# B&R Automation Studio project RS15_RX_30005_r00 (part 6)

#### BackUpCyclic.st - Cyclic code
```iecst
(********************************************************************
 * COPYRIGHT --
 ********************************************************************
 * Program: BackUp
 * File: BackUpCyclic.st
 * Author: pkiel
 * Created: December 11, 2009
 ********************************************************************
 * Implementation of program BackUp
 ********************************************************************)

PROGRAM _CYCLIC

	TON_0(IN := SystemBackUp_PB, PT := T#5s); 	(* Trigger File Write *)
	TON_1(IN := SystemRestore_PB, PT := T#5s); 	(* Trigger File Read *)
	TON_2(IN := NOT(bOK), PT := T#5s); 			(* Error Timer *)
	TON_3(IN := OpComplete, PT := T#5s); 		(* Operation Complete Timer *)
	TON_4(IN := FileNotFound, PT := T#5s); 		(* File Not Found Timer *)

	CASE byStep OF

			0: (**** Loop For Command Selection ****)

					IF (EDGEPOS(TON_0.Q)) THEN
						cmdSystemBackUp := 1;
						byStep := 1;
					ELSIF (EDGEPOS(TON_1.Q)) THEN
	                	cmdSystemRestore := 1;
						byStep := 1;
					END_IF

			1: (**** Try to open existing file ****)
	                (* Initialize file open structrue *)
	                FOpen.enable    := 1;
	                FOpen.pDevice   := ADR(strDevice);
	                FOpen.pFile     := ADR(strFile);
	                FOpen.mode      := FILE_RW;  (* Read and write access *)

	                (* Call FBK *)
	                FOpen();

	                (* Get FBK output information *)
	                dwIdent := FOpen.ident;
	                wStatus := FOpen.status;

	                (* Verify status (20708 -> File doesn't exist) *)
	                IF (wStatus = 20708) THEN
	                        IF cmdSystemBackUp THEN
									byStep := 2;
							ELSIF cmdSystemRestore THEN
	                        		byStep := 11;
							END_IF
	                ELSE
	                        IF (wStatus = 0) THEN
	                            IF cmdSystemBackUp THEN
									byStep := 3;
								ELSIF cmdSystemRestore THEN
	                        		byStep := 4;
								END_IF
	                        ELSE
	                                IF (wStatus <> 65535) THEN
	                                        byErrorLevel := 1;
	                                        byStep := 10;

	                                        IF (wStatus = 20799) THEN
	                                                wError := FileIoGetSysError();
	                                        END_IF
	                                END_IF
	                        END_IF
	                END_IF

	        2: (**** Create file ****)
	                (* Initialize file create structure *)
	                FCreate.enable  := 1;
	                FCreate.pDevice := ADR(strDevice);
	                FCreate.pFile   := ADR(strFile);

	                (* Call FBK *)
	                FCreate();

	                (* Get FBK output information *)
	                dwIdent := FCreate.ident;
	                wStatus := FCreate.status;

	                (* Verify status *)
	                IF (wStatus = 0) THEN
							byStep := 3;
	                ELSE
	                        IF (wStatus <> 65535) THEN
	                                byErrorLevel := 2;
	                                byStep := 10;

	                                IF (wStatus = 20799) THEN
	                                        wError := FileIoGetSysError();
	                                END_IF
	                        END_IF
	                END_IF

	        3: (**** Write data to file ****)
	                (* Load Data Into System Structure *)
					SystemData.gSP_A	 				        := gSP_A;
					SystemData.gReg 					        := gReg;
					SystemData.gPassword 				      := gPassword;
					SystemData.gMachineTime				    := gMachineTime;
					SystemData.gSP_CmdSpeed				    := gSP_CmdSpeed;
					SystemData.gSP_ColdGlue				    := gSP_ColdGlue;
					SystemData.gSP_HotGlue				    := gSP_HotGlue;
					SystemData.gSP_GlueTrayAutoSpeed	:= gSP_GlueTrayAutoSpeed;
					SystemData.gSP_PerfCylSelect		  := gSP_PerfCylSelect;
					SystemData.gSP_PerfKnifeCount		  := gSP_PerfKnifeCount;
					SystemData.gSP_TubeSelect		  	  := gSP_TubeSelect;

					(* Write System Structure To File *)
	                FWrite.enable   := 1;
	                FWrite.ident    := dwIdent;
	                FWrite.offset   := 0;
	                FWrite.pSrc     := ADR(SystemData);
	                FWrite.len      := SIZEOF(SystemData);

	                (* Call FBK *)
	                FWrite();

	                (* Get status *)
	                wStatus := FWrite.status;

	                (* Verify status *)
	                IF (wStatus = 0) THEN
	                        byStep := 5;
	                ELSE
	                        IF (wStatus <> 65535) THEN
	                                byErrorLevel := 3;
	                                byStep := 10;

	                                IF (wStatus = 20799) THEN
	                                        wError := FileIoGetSysError();
	                                END_IF
	                        END_IF
	                END_IF

	        4: (**** Read data from file ****)
	                (* Initialize file read structure *)
	                FRead.enable    := 1;
	                FRead.ident     := dwIdent;
	                FRead.offset    := 0;
	                FRead.pDest     := ADR(SystemData);
	                FRead.len       := SIZEOF(SystemData);

	                (* Call FBK *)
	                FRead();

	                (* Get status *)
	                wStatus := FRead.status;

	                (* Verify status *)
	                IF (wStatus = 0) THEN
						gSP_A 						    := SystemData.gSP_A;
						gReg 					      	:= SystemData.gReg;
						gPassword 					  := SystemData.gPassword;
						gMachineTime				  := SystemData.gMachineTime;
						gSP_CmdSpeed				  := SystemData.gSP_CmdSpeed;
						gSP_ColdGlue	 			  := SystemData.gSP_ColdGlue;
						gSP_HotGlue					  := SystemData.gSP_HotGlue;
						gSP_GlueTrayAutoSpeed	:= SystemData.gSP_GlueTrayAutoSpeed;
						gSP_PerfCylSelect			:= SystemData.gSP_PerfCylSelect;
						gSP_PerfKnifeCount		:= SystemData.gSP_PerfKnifeCount;
						gSP_TubeSelect				:= SystemData.gSP_TubeSelect;

						byStep := 5;
	                ELSE
	                    IF (wStatus <> 65535) THEN
	                 	   byErrorLevel := 4;
	                       byStep := 10;

	                       IF (wStatus = 20799) THEN
	                    	   wError := FileIoGetSysError();
	                       END_IF
	                	END_IF
	                END_IF

	        5: (**** Close file ****)
	                (* Initialize file close structure *)
	                FClose.enable   := 1;
	                FClose.ident    := dwIdent;

	                (* Call FBK *)
	                FClose();

	                (* Get status *)
	                wStatus := FClose.status;

	                (* Verify status *)
	                IF (wStatus = 0) THEN
							cmdSystemBackUp := 0;
							cmdSystemRestore := 0;
	                        OpComplete := 1;
							byStep := 6;
	                ELSE
	                        IF (wStatus <> 65535) THEN
	                                byErrorLevel := 5;
	                                byStep := 10;

	                                IF (wStatus = 20799) THEN
	                                        wError := FileIoGetSysError();
	                                END_IF
	                        END_IF
	                END_IF

	        6: (**** Operation Complete ****)

	                IF (TON_3.Q) THEN
						OpComplete := 0;
						byStep := 0;
					END_IF

			10: (**** Error step ****)
	                bOK := FALSE;
					cmdSystemBackUp := 0;
					cmdSystemRestore := 0;
					IF (TON_2.Q) THEN
						bOK := 1;
						byStep := 0;
					END_IF

			11: (**** File Not Found ****)
	                bOK := FALSE;
					FileNotFound := 1;
					cmdSystemBackUp := 0;
					cmdSystemRestore := 0;
	                IF (TON_4.Q) THEN
						FileNotFound := 0;
						bOK := TRUE;
						byStep := 0;
					END_IF

	END_CASE

END_PROGRAM
```

#### BackUp.var - Local variables
```iecst
(********************************************************************
 * COPYRIGHT --
 ********************************************************************
 * Program: BackUp
 * File: BackUp.var
 * Author: pkiel
 * Created: December 11, 2009
 ********************************************************************
 * Local variables of program BackUp
 ********************************************************************)
VAR
	strDevice : STRING[32];
	strFile : STRING[32];
	byStep : USINT;
	FOpen : FileOpen;
	bOK : BOOL;
	dwIdent : UDINT;
	wStatus : UINT;
	byErrorLevel : USINT;
	wError : UINT;
	FCreate : FileCreate;
	FWrite : FileWrite;
	FRead : FileRead;
	FClose : FileClose;
	TON_0 : TON;
	TON_1 : TON;
	TON_2 : TON;
	TON_3 : TON;
	TON_4 : TON;
	OpComplete : BOOL;
	SystemBackUp_PB : BOOL;
	SystemRestore_PB : BOOL;
	cmdSystemBackUp : BOOL;
	cmdSystemRestore : BOOL;
	FileNotFound : BOOL;
	SystemData : System;
END_VAR
```

- Program Logical/HMI/Cmd_Trace (IEC) (no source held here)

### Program Logical/HMI/CPURestart

#### CPURestartCyclic.st
```iecst
(********************************************************************
 * COPYRIGHT -- .
 ********************************************************************
 * Program: CPURestart
 * File: CPURestartCyclic.st
 * Author: dominique
 * Created: March 18, 2012
 ********************************************************************
 * Implementation of program CPURestart
 ********************************************************************)

PROGRAM _CYCLIC

  // Sytem Restart from HMI

  // Cold
  IF HMI_CmdColdRestart THEN
    HMI_CmdColdRestart := 0 ;
    uiRetColdRestart := SYSreset(1, 2) ;
    IF (uiRetColdRestart <> 0) THEN
      HMI_iCRestartStat := uiRetColdRestart ;
    END_IF
  END_IF

  // Warm
  IF HMI_CmdWarmRestart THEN
    HMI_CmdWarmRestart := 0 ;
    uiRetWarmRestart := SYSreset(1, 1) ;
    IF (uiRetWarmRestart <> 0) THEN
      HMI_iWRestartStat := uiRetWarmRestart ;
    END_IF
  END_IF

  // Reset stat
  IF EDGEPOS(gAlarmReset) THEN
    HMI_iCRestartStat := 0 ;
    HMI_iWRestartStat := 0 ;
  END_IF

END_PROGRAM
```

#### CPURestartInit.st
```iecst
(********************************************************************
 * COPYRIGHT -- .
 ********************************************************************
 * Program: CPURestart
 * File: CPURestartInit.st
 * Author: dominique
 * Created: March 18, 2012
 ********************************************************************
 * Implementation of program CPURestart
 ********************************************************************)

PROGRAM _INIT

END_PROGRAM
```

- FreeLock.clm (not shown)

- GreenRed.clm (not shown)

- Sensor.clm (not shown)

- SetCol_1.clm (not shown)

- Arial10pxBold.fninfo (not shown)

- Arial12px.fninfo (not shown)

- Arial9pxBold.fninfo (not shown)

- Arial_12_Bold.fninfo (not shown)

- Arial_12_Bold_Italic.fninfo (not shown)

- Arial_14_Bold_Italic.fninfo (not shown)

- Arial_15_Bold.fninfo (not shown)

- Arial_18_Bold.fninfo (not shown)

- Arial_18_Italic.fninfo (not shown)

- Arial_20_Bold.fninfo (not shown)

- Arial_26_Bold.fninfo (not shown)

- Arial_36_Bold.fninfo (not shown)

- Arial_8_Bold.fninfo (not shown)

- Arial_9_Bold.fninfo (not shown)

- EnvBagPerfSetUp.layer (not shown)

- PasswordChangeAccepted.layer (not shown)

- PasswordConfirm.layer (not shown)

- PerfSpeedCurve_RS15_Perfo1_2_IF.layer (not shown)

- PerfSpeedCurve_RS26_ApPo_520_IF.layer (not shown)

- PerfSpeedCurve_RS26_Perfo1_IF.layer (not shown)

- PopUp_AxisSynchroInProgress.layer (not shown)

- PopUp_ProductCountReset.layer (not shown)

- SetUpHoldTearApPoDrumRS26.layer (not shown)

- StandPerfSetUp.layer (not shown)

- Underlay_Alarms.layer (not shown)

- Underlay_Main.layer (not shown)

- Underlay_Maintenance.layer (not shown)

- Underlay_Setup.layer (not shown)

- ZZZ.layer (not shown)

- TrendData_1.trd (not shown)

- TrendData_2.trd (not shown)

### Program Logical/HMI/HMI_Control

#### HMI_Control.var
```iecst
(********************************************************************
 * COPYRIGHT --
 ********************************************************************
 * Program: HMI_Control
 * File: HMI_Control.var
 * Author: pkiel
 * Created: September 17, 2009
 ********************************************************************
 * Local variables of program HMI_Control
 ********************************************************************)
VAR
	CfgSetDefaultGateway_0 : CfgSetDefaultGateway;
	DataLock_Motion : UINT;
	HMI_ActualVelocity : REAL;
	HMI_AlarmFilterControl : INT;
	HMI_AlarmFilterGroup : INT;
	HMI_AlarmInputStatus : INT;
	HMI_Error : BOOL;
	HMI_ErrorAck : BOOL;
	HMI_ErrorCount : UINT;
	HMI_ErrorID : UINT;
	HMI_ErrorStop : BOOL;
	HMI_ErrorText : ARRAY[0..3] OF STRING[79];
	HMI_Ind_ContinuousMotion : BOOL;
	HMI_Ind_ControllerStatus : BOOL;
	HMI_Ind_DiscreteMotion : BOOL;
	HMI_Ind_Enabled : BOOL;
	HMI_Ind_Homed : BOOL;
	HMI_Ind_InMotion : BOOL;
	HMI_Ind_NetworkInit : BOOL;
	HMI_Ind_SynchronizedMotion : BOOL;
	HMI_Input_DriveEnable : BOOL;
	HMI_Input_Home : BOOL;
	HMI_Input_Trigger1 : BOOL;
	HMI_Input_Trigger2 : BOOL;
	HMI_MainScreenGroup : UINT;
	HMI_MaintenanceScreenGroup : UINT;
	HMI_PositionDeg : REAL;
	HMI_PositionInch : REAL;
	HMI_Screen2Group_Ind : UINT;
	HMI_ScreenGroup_Ind : UINT;
	HMI_SetupScreenGroup : UINT;
	HMI_Status_Ind : UINT;
	HMI_StatusScreenGroup : UINT;
	HMI_bMaxSpeedPerf_PB : BOOL;
	HMI_iSelCurvMaxSpeedPerf : INT;
	HMI_uiCurvVisibl : UINT;
	HMI_uiNeverVisibl : UINT := 1;
	HMI_strMP_UNW_HydroPump : STRING[10];
	HMI_strMP_FP_MotorFan : STRING[10];
	HMI_strMP_FP_SlowRot1 : STRING[10];
	HMI_strMP_FP_SlowRot2 : STRING[10];
	HMI_strMP_FP_SlowRot3 : STRING[10];
	HMI_strMP_FP_SlowRot4 : STRING[10];
	HMI_strMP_FP_SlowRot5 : STRING[10];
	HMI_strMP_FP_SlowRot6 : STRING[10];
	HMI_strMP_GlueSlowRotation : STRING[10];
	HMI_strMP_PerfFan : STRING[10];
	HMI_strMP_Vacuum : STRING[10];
	HMI_strMP_3W_MotorFan : STRING[10];
	HMI_strMP_DRY_Blower : STRING[12];
	HMI_strMP_DRY_Heater : STRING[10];
	HMI_strSS_DRY_Thermostat : STRING[10];
	HMI_strMP_CMP_WasteSuc : STRING[10];
	HMI_strMP_EB_WasteSuc : STRING[10]; (*Envelope Bag Waste Suction*)
	HMI_iAnimHoldTearEnvB_1 : INT;
	HMI_iAnimHoldTearEnvB_2 : INT;
	HMI_iNumbPliers_1 : INT;
	HMI_iNumbPliers_2 : INT;
	HMI_iAnimPictHoldTearEnvB : INT;
	HMI_bPBShowEnvBConf : BOOL;
	HMI_rTubLInf_1 : REAL;
	HMI_rTubLInf_2 : REAL;
	HMI_rTubLSup_1 : REAL;
	HMI_rTubLSup_2 : REAL;
	HMI_iAnimPict2Visibl : INT;
	HMI_iAnimTubLVisibl : INT;
	HMI_rPosHoldEnvB : REAL;
	rPosHoldEnvB : REAL;
	HMI_iAnimSynchroAxis : INT;
	HMI_iAnimSynchroAxisVisibl : INT;
	HMI_iHTEnvBOffsetVisibl : INT;
	iAnimStep : INT;
	iCountCycl : INT;
	iIndex : INT;
	Count : INT;
END_VAR
```

#### HMI_ControlCyclic.st
```iecst
(********************************************************************
 * COPYRIGHT --
 ********************************************************************
 * Program: HMI_Control
 * File: HMI_ControlCyclic.st
 * Author: pkiel
 * Created: September 17, 2009
 ********************************************************************
 * Implementation of program HMI_Control
 ********************************************************************)

PROGRAM _CYCLIC
//		IF gPowerUp_Complete AND (Count<5) THEN
//			gA[0].ErrorAck := 1;
//			Count := Count + 1;
//		END_IF

(* Screen GoTo Control on Main HMI For Main, Setup, & Status Screens *)
	IF (gHMI_GoToMain_PB) THEN
		gScreenControl:=HMI_MainScreenGroup;
		gHMI_GoToMain_PB:=0;
		HMI_ScreenGroup_Ind:=0;
		gHMI_PasswordLevel:=0;
	END_IF;
	IF (gHMI_GoToSetup_PB) THEN
		gScreenControl:=HMI_SetupScreenGroup;
		gHMI_GoToSetup_PB:=0;
		HMI_ScreenGroup_Ind:=1;
		gHMI_PasswordLevel:=0;
	END_IF;
	IF (gHMI_GoToStatus_PB) THEN
		gScreenControl:=20;
		gHMI_GoToStatus_PB:=0;
		HMI_ScreenGroup_Ind:=2;
		gHMI_PasswordLevel:=0;
	END_IF;
	IF (gHMI_GoToAlarm_PB) THEN
		gScreenControl:=30;
		gHMI_GoToAlarm_PB:=0;
		HMI_ScreenGroup_Ind:=4;
		gHMI_PasswordLevel:=0;
	END_IF;
  IF (gHMI_GoToMaint_PB) THEN
    gScreenControl:=HMI_MaintenanceScreenGroup;
    gMaintDropdown := gScreenControl;
    gHMI_GoToMaint_PB:=0;
    HMI_ScreenGroup_Ind:=3;
  END_IF;
  IF (gHMI_GoToHoldTearDrum_PB) THEN
    gScreenControl:=12;
    gHMI_GoToHoldTearDrum_PB:=0;
  END_IF;
	CASE (HMI_ScreenGroup_Ind) OF
		0:
			HMI_MainScreenGroup:=gCurrentScreen;
			HMI_MainScreenGroup:=LIMIT(1,HMI_MainScreenGroup,6);
		1:
			HMI_SetupScreenGroup:=gCurrentScreen;
			HMI_SetupScreenGroup:=LIMIT(10,HMI_SetupScreenGroup,12);

		2:
			HMI_StatusScreenGroup:=gCurrentScreen;
			HMI_StatusScreenGroup:=LIMIT(20,HMI_StatusScreenGroup,20);
		3:
			IF (gMaintScreenChange) THEN
				gScreenControl := gMaintDropdown;
				gMaintScreenChange :=0;
			END_IF
			HMI_MaintenanceScreenGroup:=gCurrentScreen;
			HMI_MaintenanceScreenGroup:=LIMIT(40,HMI_MaintenanceScreenGroup,57);
	END_CASE;

(* Transfers for Servo Status Screens *)
	HMI_Status_Ind:=LIMIT(0,HMI_Status_Ind,15);
	IF (gCurrentScreen=20) THEN
			gA[HMI_Status_Ind].ErrorAck			:=	HMI_ErrorAck;
			HMI_ErrorCount				:=	gA[HMI_Status_Ind].ErrorCount;
			HMI_ErrorText				:=	gA[HMI_Status_Ind].ErrorText;
			HMI_Ind_Enabled				:=	gA[HMI_Status_Ind].Ind_Enabled;
			HMI_Ind_InMotion			:=	gA[HMI_Status_Ind].Ind_InMotion;
			HMI_Error					:=	gA[HMI_Status_Ind].Error;
			HMI_ErrorStop				:=	gA[HMI_Status_Ind].ErrorStop;
			HMI_ErrorID					:=	gA[HMI_Status_Ind].ErrorID;
			HMI_Ind_DiscreteMotion		:=	gA[HMI_Status_Ind].Ind_DiscreteMotion;
			HMI_Ind_ContinuousMotion	:=	gA[HMI_Status_Ind].Ind_ContinuousMotion;
			HMI_Ind_SynchronizedMotion	:=	gA[HMI_Status_Ind].Ind_SynchronizedMotion;
			HMI_Ind_NetworkInit			:=	gA[HMI_Status_Ind].Ind_NetworkInit;
			HMI_Ind_ControllerStatus	:=	gA[HMI_Status_Ind].Ind_ControllerStatus;
			HMI_Ind_Homed				:=	gA[HMI_Status_Ind].Ind_Homed;
			HMI_Input_Home				:=	gA[HMI_Status_Ind].Input_Home;
			HMI_Input_DriveEnable		:=	gA[HMI_Status_Ind].Input_DriveEnable;
			HMI_Input_Trigger1			:=	gA[HMI_Status_Ind].Input_Trigger1;
			HMI_Input_Trigger2			:=	gA[HMI_Status_Ind].Input_Trigger2;
			HMI_PositionInch			:=	gA[HMI_Status_Ind].PositionInch;
			HMI_PositionDeg				:=	gA[HMI_Status_Ind].PositionDeg;
			HMI_ActualVelocity			:=	gA[HMI_Status_Ind].ActualVelocity;
	END_IF

(*Data Entry Lockout*)
	IF (gA[9].Ind_InMotion) THEN
		DataLock_Motion := 2;
  ELSE
    DataLock_Motion := 0;
	END_IF

// Display curve max speed Perf
  IF HMI_bMaxSpeedPerf_PB THEN
    HMI_iSelCurvMaxSpeedPerf := gInchMetric_Ind ;
    HMI_uiCurvVisibl := 0 ; // Curve visible
  ELSE
    HMI_iSelCurvMaxSpeedPerf := 0 ;
    HMI_uiCurvVisibl := 1 ; // Curve unvisible
  END_IF
  IF (gCurrentScreen <> 11) THEN
    HMI_bMaxSpeedPerf_PB := 0 ;
  END_IF

// Hide Holding Tearing Envelope Bag Offset
  IF (gCurrentScreen <> 1) THEN
    HMI_iHTEnvBOffsetVisibl := 1 ;
  END_IF

// ----------------------------------------------------------------------------------------
// Picture animation

    // Sychro axis animation
    IF g_bSynchroAxisInProgress THEN
      iCountCycl := iCountCycl + 1 ;
      IF (iCountCycl >= 3) THEN      // HMI_Control Task time = 0,1s. Animation => 25 pictures/s => Cycle count >= 2.5 (=>3)
        iCountCycl := 0 ;
        iAnimStep  := iAnimStep + 1 ;
        HMI_iAnimSynchroAxis := iAnimStep ;
        IF (iAnimStep >= 4) THEN
          iAnimStep := 0 ;
        END_IF
      END_IF
      HMI_iAnimSynchroAxisVisibl := 0 ;    // Visible
    ELSE
      iCountCycl := 0 ;
      iAnimStep  := 0 ;
      HMI_iAnimSynchroAxis := 0 ;
      HMI_iAnimSynchroAxisVisibl := 1 ;    // Not visible
    END_IF

    // Help view axis config
    IF NOT(HMI_bPBShowEnvBConf) THEN
      IF HMI_iAnimPictHoldTearEnvB > 2 THEN
        HMI_iAnimPictHoldTearEnvB := 1 ;
      END_IF
      IF HMI_iAnimPictHoldTearEnvB < 1 THEN
        HMI_iAnimPictHoldTearEnvB := 2 ;
      END_IF
      HMI_iAnimTubLVisibl := 0 ; // Visible

      CASE HMI_iAnimPictHoldTearEnvB OF
        1 :
          HMI_iAnimHoldTearEnvB_1 := 1 ;
          HMI_iAnimHoldTearEnvB_2 := 2 ;
          HMI_rTubLInf_1 := g_rMinBagSize_RS26_mm/25.4 ;
          HMI_rTubLSup_1 := gr_rBagSize4_2Pliers_mm/25.4 ;
          HMI_rTubLInf_2 := gr_rBagSize4_2Pliers_mm/25.4 ;
          HMI_rTubLSup_2 := gr_rEnvBSizeTear2_1_mm/25.4 ;
          HMI_iNumbPliers_1 := 4 ;
          HMI_iNumbPliers_2 := 2 ;
          HMI_iAnimPict2Visibl := 0 ;
        2 :
          HMI_iAnimHoldTearEnvB_1 := 3 ;
          HMI_iAnimHoldTearEnvB_2 := 0 ;
          HMI_rTubLInf_1 := gr_rEnvBSizeTear2_1_mm/25.4 ;
          HMI_rTubLSup_1 := g_rMaxBagSize_RS26_mm/25.4 ;
          HMI_rTubLInf_2 := 0.0 ;
          HMI_rTubLSup_2 := 0.0 ;
          HMI_iNumbPliers_1 := 2 ;
          HMI_iNumbPliers_2 := 0 ;
          HMI_iAnimPict2Visibl := 1 ; // Hide
      END_CASE
      rPosHoldEnvB := gr_rPosEnvBHoldBag + 45.0 ;
      HMI_rPosHoldEnvB := H_FC_Modulus (
                               IN_rMod := 360.0 ,
                               IN_rVar := rPosHoldEnvB
                                       ) ;
    ELSE
      HMI_iAnimTubLVisibl     := 1 ; // Hide
      HMI_iAnimHoldTearEnvB_1 := 4 ;
      HMI_iAnimHoldTearEnvB_2 := 5 ;
      HMI_rTubLInf_1 := g_rMinBagSize_EnvB_mm/25.4 ;
      HMI_rTubLSup_1 := gr_rBagSize1_2Hold_mm/25.4 ;
      HMI_rTubLInf_2 := gr_rBagSize1_2Hold_mm/25.4 ;
      HMI_rTubLSup_2 := g_rMaxBagSize_EnvB_mm/25.4 ;
      HMI_iNumbPliers_1 := 2 ;
      HMI_iNumbPliers_2 := 2 ;
      HMI_iAnimPict2Visibl := 0 ;
      HMI_rPosHoldEnvB := gr_rPosEnvBHoldBag ;
    END_IF

END_PROGRAM
```

#### HMI_ControlInit.st
```iecst
(********************************************************************
 * COPYRIGHT --
 ********************************************************************
 * Program: HMI_Control
 * File: HMI_ControlInit.st
 * Author: pkiel
 * Created: September 17, 2009
 ********************************************************************
 * Implementation of program HMI_Control
 ********************************************************************)

PROGRAM _INIT

	HMI_MainScreenGroup:=1;
	HMI_SetupScreenGroup:=10;
	HMI_StatusScreenGroup:=20;
	HMI_MaintenanceScreenGroup:=40;
	HMI_AlarmInputStatus:=HMI_AlarmInputStatus;
  HMI_uiCurvVisibl := 1 ;
  HMI_uiNeverVisibl := 1 ;

  // Unwinder
  HMI_strMP_UNW_HydroPump    := '21Q1' ;
  // Flexo Press
  HMI_strMP_FP_MotorFan      := '73Q2' ;
  HMI_strMP_FP_SlowRot1      := '27Q1' ;
  HMI_strMP_FP_SlowRot2      := '27Q2' ;
  HMI_strMP_FP_SlowRot3      := '27Q3' ;
  HMI_strMP_FP_SlowRot4      := '27Q4' ;
  HMI_strMP_FP_SlowRot5      := '28Q1' ;
  HMI_strMP_FP_SlowRot6      := '28Q2' ;
  // Bag Machine
  HMI_strMP_GlueSlowRotation := '19Q1' ;
  HMI_strMP_PerfFan          := '73Q4' ;
  HMI_strMP_Vacuum           := '14Q1' ;
  // 3-Web unit
  HMI_strMP_3W_MotorFan      := '36Q1' ;
  // Dryer
  HMI_strMP_DRY_Blower       := '31Q1 OR 31Q2' ;
  HMI_strMP_DRY_Heater       := '3Q5' ;
  HMI_strSS_DRY_Thermostat   := '79F1' ;
  // Cold Micro Perf Waste suction
  HMI_strMP_CMP_WasteSuc     := '15Q2' ;
  // Envelope Bag Waste Suction
  HMI_strMP_EB_WasteSuc      := '36Q1' ;

  HMI_iAnimSynchroAxisVisibl := 1 ;
  g_bSplashDone := 0 ;

  HMI_iHTEnvBOffsetVisibl := 1 ;

	// Initialize Default Gateway...RS26 Pyrollpack_14661 IP Config IP Adresse  : 10.0.1.67
  //                                                               Gateway    : 10.0.1.1
  //                                                               SubNetMask : 255.255.255.0
	CfgSetDefaultGateway_0(enable := 1 , pDevice := ADR('IF5'), pGateway := ADR('10.0.1.1'), Option := 1);

	// Make Sure Values Are Initialized
	g_rBagSize1to2SPerf_mm		:= 190.0;
	g_rBagSize1to2LPerf_mm		:= 260.0;
	g_rLinSpeedMin_mmin			:= 10.0;
	g_rMaxSpeedMin_bpm			:= 35.0;
	g_rMaxSpeedSynchro_bpm		:= 8.0;
	g_rMaxJogDecel_bpmm			:= 1200.0;
	g_rLinSpeedSP_AccRS26		:= 600.0;
	g_rLinSpeedSP_DecRS26		:= 600.0;
	g_rLinSpeedSP_JogDecRS26	:= 2500.0;
	g_rLinSpeedSP_EStopDecRS26	:= 6000.0;
	g_rLinSpeedSP_GuardFaultDecRS26 := 4500.0;
	g_rLinSpeedSP_WebBreakDecRS26 := 5200.0;
	g_rLinSpeedSP_GenFaultDecRS26 := 3000.0;
	g_rLinSpeedSP_FStopDecRS26	:= 1800.0;
	g_rLinSpeedSP_AccRS15		:= 33.3;
	g_rLinSpeedSP_DecRS15		:= 33.3;
	g_rLinSpeedSP_JogDecRS15	:= 140.0;
	g_rLinSpeedSP_EStopDecRS15	:= 333.0;
	g_rLinSpeedSP_GuardFaultDecRS15 := 250.0;
	g_rLinSpeedSP_WebBreakDecRS15 := 250.0;
	g_rLinSpeedSP_GenFaultDecRS15 := 167.0;
	g_rLinSpeedSP_FStopDecRS15	:= 100.0;
	g_rSizeEntryPullRol_mm		:= 400.0;
	g_rSizeExitPullRol_mm		:= 320.0;
	g_rSizeLPerf_mm				:= 400.0;
	g_rSizeSPerf_mm				:= 270.0;
	g_rSizeDrum_mm				:= 1680.0;
	g_rZGearRepFP_M				:= 40.0;
	g_rZGearRepFP_8DP			:= 40.0;
	g_rZGearRepFP_10DP			:= 50.0;
	g_rZGearRepFP_1_4P			:= 65.0;
	g_rZGearCMPerf_M			:= 50.0;
	g_rZGearCMPerf_8DP			:= 50.0;
	g_rZGearCMPerf_10DP			:= 63.0;
	g_rZGearCMPerf_1_4P			:= 81.0;
	g_rMaxBagSize_RS15_mm		:= 400.0;
	g_rMinBagSize_RS15_mm		:= 105.0;
	g_rMaxBagSize_RS26_mm		:= 760.0;
	g_rMinBagSize_RS26_mm		:= 160.0;
	g_rMaxBagSize_EnvB_mm		:= 760.0;
	g_rMinBagSize_EnvB_mm		:= 240.0;
	g_rSizeEnvBPerf_mm			:= 520.0;
	gr_rMachMaxSpeed_BPM		:= 1000.0;
	gr_rHoldAxContactZone		:= 22.0;
	gr_rTearAxContactZone		:= 52.0;
	gr_rDrumAxContactZone		:= 50.0;
	gr_rEnvBAxContactZone		:= 26.0;
	gr_rTearEBAxContactZone		:= 52.0;
	gr_rPosHoldBag				:= 11.0;
	gr_rPosTearBag				:= 26.0;
	gr_rPosGripBag				:= 25.0;
	gr_rPosEnvBHoldBag			:= 355.0;
	gr_rPosTearEBTearBag		:= 18.0;
	gr_rAxisTimSet_SP_Vel		:= 12.0;
	gr_rAxisTimSet_SP_Acc		:= 1200.0;
	gr_rAxisTimSet_SP_Dec		:= 3000.0;
	gr_rMaxRangeWebDraw			:= 1.0;
	gr_rLimOffsetRunVal			:= 0.1;
	gr_rIncrOffsetAxeRun		:= 1.0;
	gr_tJogHornDur				:= T#1s;
	gr_tRunHornDur				:= T#1500ms;
	gr_rMaxLSFlexoP_mmin		:= 300.0;
	gr_rDistPerfTearEnvBOn_mm	:= 4560.0;
	gr_rDistPerfTearEnvBOff4_mm := 4260.0;
	gr_rDistPerfTearEnvBOff2_mm	:= 4560.0;
	gr_rSizeEnvBLowRol_mm		:= 440.0;
	gr_rTearCarStep_mm			:= 413.0;
	gr_rDistPerfTearRS26_mm		:= 3800.0;
	gr_rDistPerfTearRS15_mm		:= 3700.0;
	gr_rIncrShiftPerf_mm		:= 1.0;
	gr_rBagSize2_4Hold_mm		:= 160.0;
	gr_rBagSize1_2Hold_mm		:= 320.0;
	gr_rBagSize4_2Pliers_mm		:= 400.0;
	gr_rEnvBSizeTear2_1_mm		:= 500.0;
	gr_rHMPerfSlowRot_rpm		:= 2.0;
	gr_rHMPerfAcc_rpm2			:= 120.0;
	gr_rHMPerfDec_rpm2			:= 5000.0;
	gr_rHMPerfSlowRot_rpm		:= 2.0;
	gr_rHMPerfAcc_rpm2			:= 120.0;
	gr_rHMPerfDec_rpm2 			:= 5000.0;
	gr_rHMPerfSLActTool_mmin	:= 20;

END_PROGRAM
```

### Program Logical/HMI/Language

#### LanguageCyclic.st
```iecst
(********************************************************************
 * COPYRIGHT --
 ********************************************************************
 * Program: Language
 * File: LanguageCyclic.st
 * Author: pkiel
 * Created: October 09, 2009
 ********************************************************************
 * Implementation of program Language
 ********************************************************************)

PROGRAM _CYCLIC

(*Language Control*)
	IF (Language_PB=0) THEN
		Language_Ind := 0;
	ELSE
		Language_Ind := 2; // Fr
	END_IF

END_PROGRAM
```

- Program Logical/HMI/Message_1 (IEC) (no source held here)

- Program Logical/HMI/Message_2 (IEC) (no source held here)

### Program Logical/HMI/Password (IEC)

#### PasswordInit.st - Initialization code
```iecst
(********************************************************************
 * COPYRIGHT --
 ********************************************************************
 * Program: Password
 * File: PasswordInit.st
 * Author: pkiel
 * Created: October 20, 2009
 ********************************************************************
 * Implementation of program Password
 ********************************************************************)

PROGRAM _INIT

	UserLevel_Ind := 0;
	PasswordStatus := 0;
	InvalidPassword_Ind := 1;
//	IF (NOT FirstBoot) THEN
		gPassword.Supervisor  := 'super';
		gPassword.Maintenance := 'maint';
		gPassword.Technician  := 'tech725';
//		FirstBoot := 1;
//	END_IF
	PasswordAccepted_Visibility := 1;
	PasswordChange_Visibility := 1;
	PasswordFail_Visibility := 1;
  PasswordConfirm_Visibility := 1;

  iDryerTrend_Visibility := 1 ;

END_PROGRAM
```

#### Password.var - Local variables
```iecst
(********************************************************************
 * COPYRIGHT --
 ********************************************************************
 * Program: Password
 * File: Password.var
 * Author: pkiel
 * Created: October 20, 2009
 ********************************************************************
 * Local variables of program Password
 ********************************************************************)
VAR
	CurrentUser : STRING[32];
	DataLock_0 : UINT;
	DataLock_1 : UINT;
	DataLock_2 : UINT;
	DataLock_3 : UINT;
	UserLevel_Ind : UINT;
	PasswordStatus : UINT;
	EvaluatePassword : BOOL := FALSE;
	PasswordEntered : STRING[32];
	InvalidPassword : BOOL := FALSE;
	Logout_PB : BOOL;
	TON_0 : TON;
	InvalidPassword_Ind : UINT;
	PasswordChange_Visibility : UINT;
	PasswordNew : STRING[32];
	PasswordConfirm : STRING[32];
	StringLength : INT;
	PasswordSelect_Ind : UINT;
	PasswordChangeFailure : BOOL;
	PasswordChangeAccepted : BOOL;
	PasswordAccepted_Visibility : UINT;
	TON_1 : TON;
	PasswordFail_Visibility : UINT;
	TON_2 : TON;
	PasswordChangeCancel_PB : BOOL;
	PasswordChangeAccept_PB : BOOL;
	PasswordChangeStart_PB : BOOL;
  PasswordConfirm_Visibility : UINT;
  iDryerTrend_Visibility : INT ;
END_VAR
VAR RETAIN
	FirstBoot : BOOL;
END_VAR
```

- Program Logical/HMI/Recipe_1 (IEC) (no source held here)

### Program Logical/HMI/Recipe_2 (IEC)

#### Recipe_2.var - Local variables
```iecst
(********************************************************************
 * COPYRIGHT --
 ********************************************************************
 * Program: Recipe_2
 * File: Recipe_2.var
 * Author: pkiel
 * Created: November 16, 2009
 ********************************************************************
 * Local variables of program Recipe_2
 ********************************************************************)
VAR CONSTANT
	INIT_STEP : UINT := 000;
	INIT_WAIT : UINT := 005;
	INIT_RECIPE : UINT := 010;
	ERROR_STEP : UINT := 200;
	MAX_RECIPE : UDINT := 200;
	COMMAND_RECIPE : UINT := 050;
	DELETE_RECIPE : UINT := 060;
	LOAD_RECIPE : UINT := 080;
	SAVE_RECIPE : UINT := 070;
	CR : USINT := 13;
	SPACE : USINT := 32;
END_VAR
VAR
	CSV_Init_0 : CSV_Init;
	pNames : ARRAY[0..9] OF UDINT;
	step : UINT;
	pDevice : ARRAY[0..9] OF UDINT;
	recipeName : ARRAY[0..199] OF STRING[20];
	indexNum : UINT;
	DirCreate_0 : DirCreate;
	waitCnt : UINT;
	wError : UINT;
	errStep : UINT;
	errorLevel : USINT;
	DirInfo_0 : DirInfo;
	dirNum : UDINT;
	fileNum : UDINT;
	readDir : fiDIR_READ_DATA;
	fileCounter : UDINT;
	recipeDescription : ARRAY[0..199] OF STRING[80];
	DirRead_0 : DirRead;
	stsCnt : UINT;
	FileOpen_0 : FileOpen;
	FileRead_0 : FileRead;
	strLenChk : UDINT;
	FileClose_0 : FileClose;
	pDeviceDir : UDINT;
	driveSelectOld : USINT;
	tempString : STRING[80];
	FileDelete_0 : FileDelete;
	FileWrite_0 : FileWrite;
	FileCreate_0 : FileCreate;
	errorString : STRING[80];
	CSV_Search_0 : CSV_Search;
	CSV_WriteFile_0 : CSV_WriteFile;
	CSV_ReadFile_0 : CSV_ReadFile;
	commentString : STRING[80];
	recipeDescriptionTemp : STRING[80];
	cnt : UINT;
	cr : USINT;
	deviceSelect : BOOL;
	hmiDeviceSelect : BOOL;
	hmiDevice : BOOL;
	mecChk : UDINT;
	memChk : UDINT;
	countString : STRING[10];
	totalNumString : STRING[10];
	RecipeBackUpPopUp : UINT;
	RecipeRestorePopUp : UINT;
	pChar : REFERENCE TO USINT;
END_VAR
```

### Program Logical/HMI/Splash (IEC)

#### Splash.var - Local variables
```iecst
(********************************************************************
 * COPYRIGHT --
 ********************************************************************
 * Program: Splash
 * File: Splash.var
 * Author: pkiel
 * Created: October 09, 2009
 ********************************************************************
 * Local variables of program Splash
 ********************************************************************)
VAR
	CountDown : REAL;
	CountDown2 : REAL;
	ElapsedTime : REAL;
	ElapsedTime2 : REAL;
	Ready : BOOL;
	Ready2 : BOOL;
	SplashDone : BOOL;
	SplashDone2 : BOOL;
	Status : UINT;
	Status2 : UINT;
	TON_0 : TON;
	TON_1 : TON;
	VC_HANDLE : UDINT;
	VC_HANDLE2 : UDINT;
	First : BOOL;
END_VAR
```

### Program Logical/HMI/Units (IEC)

#### UnitsCyclic.st - Cyclic code
```iecst
(********************************************************************
 * COPYRIGHT --
 ********************************************************************
 * Program: Units
 * File: UnitsCyclic.st
 * Author: pkiel
 * Created: October 09, 2009
 ********************************************************************
 * Implementation of program Units
 ********************************************************************)

PROGRAM _CYCLIC

(*Inch/Metric Control*)
	IF (InchMetric_PB=0) THEN
		gInchMetric_Ind := 1; // 1 => Inch
	ELSE
		gInchMetric_Ind := 2; // 2 => Metric
	END_IF

END_PROGRAM
```

#### UnitsInit.st - Initialization code
```iecst
(********************************************************************
 * COPYRIGHT -- .
 ********************************************************************
 * Program: Units
 * File: NewProgramInit.st
 * Author: dominique
 * Created: December 09, 2011
 ********************************************************************
 * Implementation of program Units
 ********************************************************************)

PROGRAM _INIT

  InchMetric_PB := 0 ; // Inch as default value

END_PROGRAM
```

- Program Logical/Information (IEC) (no source held here)

### Program Logical/Libraries/CSV_File

#### CSV_File.typ
```iecst
TYPE
	CSV_ListFileOption_typ : STRUCT
		SearchVarName	:STRING[80];
		FileLenToRead	:UINT;
		MaxNrLen	:USINT;
		MaxNameLen	:USINT;
	END_STRUCT;
			_csv_exfilelist_internal : STRUCT
		Step	:USINT;
		DownLines	:UINT;
		UpLines	:UINT;
		PosFirstLine	:UINT;
		FileNumOnDisk	:UINT;
		FileNumAct	:UINT;
		Offset	:UDINT;
		TmpExtension	:STRING[4];
		FileInfo	:fiDIR_READ_DATA;
		i	:UINT;
		result1	:DINT;
		result2	:DINT;
		OptionStruct	:CSV_ListFileOption_typ;
		TmpString	:ARRAY[0..50] OF USINT;
		dateandtime	:DTStructure;
		status_alloc	:UINT;
		pFileData	:UDINT;
		FileIdent	:UDINT;
		FileFound	:BOOL;
		PositionFound	:BOOL;
		FirstSeperatorFound	:BOOL;
		SecondSeperatorFound	:BOOL;
		EndPositionFound	:BOOL;
		StartPositionName	:UDINT;
		EndPositionName	:UDINT;
		CRLF	:ARRAY[0..2] OF USINT;
		InternalFileName	:ARRAY[0..254] OF USINT;
		VarNameSearch	:ARRAY[0..5] OF USINT;
		CompleteEntry	:ARRAY[0..254] OF USINT;
	END_STRUCT;
			_csv_filelist_Internal : STRUCT
		MaxFileNum	:UINT;
		EntriesOnDisp	:USINT;
		pFileDevice	:UDINT;
		pFilelist	:UDINT;
		pActName	:UDINT;
		pTeeList	:UDINT;
		Offset	:UDINT;
		MemTempOffset	:UDINT;
		TempMemLng	:UDINT;
		ListboxPos	:UINT;
		FilePosCounter	:UINT;
		FileNumAct	:UINT;
		FileNumOnDisk	:UINT;
		AllocStatus	:UINT;
	END_STRUCT;
			_csv_init_Internal : STRUCT
		PV_xgetadrStatus	:UINT;
		PV_ninfoStatus	:UINT;
		PV_itemStatus	:UINT;
		TMP_allocStatus	:UINT;
		Dimension	:UINT;
		ItemNrSoll	:ARRAY[0..49] OF UINT;
		ItemNrIst	:ARRAY[0..49] OF UINT;
		i	:UINT;
		CRLF	:ARRAY[0..2] OF USINT;
		Ebene	:USINT;
		Step	:USINT;
		FoundChar	:USINT;
		Counter_Usint	:USINT;
		NameCounter	:USINT;
		Merker	:USINT;
		MerkerArray	:ARRAY[0..49] OF BOOL;
		DataLenght	:UDINT;
		Datatyp	:UDINT;
		PV_Adress	:UDINT;
		Lenght	:UDINT;
		TmpValue	:UDINT;
		StartVarName	:ARRAY[0..79] OF USINT;
		FullStrukturName	:ARRAY[0..299] OF USINT;
		StrukturName	:ARRAY[0..299] OF USINT;
		Index	:ARRAY[0..6] OF USINT;
		VarItemName	:ARRAY[0..299] OF USINT;
		ItemName	:ARRAY[0..79] OF USINT;
		ArrayName	:ARRAY[0..79] OF USINT;
		Value	:ARRAY[0..79] OF USINT;
		UsintArray	:ARRAY[0..79] OF USINT;
		DintTime	:DINT;
		NextItemReady	:BOOL;
		ArrayStructure	:BOOL;
		ArrayVariable	:BOOL;
		VariableCounter	:UDINT;
	END_STRUCT;
			_csv_read_internal : STRUCT
		OnlyArray	:BOOL;
		OnlyArrayInStruct	:BOOL;
		DateAndTime	:BOOL;
		HeaderLine	:BOOL;
		DynamicVariable	:BOOL;
		Step	:USINT;
		NameEntered	:USINT;
		ArrayStructureStarts	:USINT;
		level	:USINT;
		TmpDateTime	:ARRAY[0..79] OF USINT;
		TmpDataTyp	:ARRAY[0..79] OF USINT;
		Value	:ARRAY[0..79] OF USINT;
		TmpName	:ARRAY[0..149] OF USINT;
		StructName	:ARRAY[0..149] OF USINT;
		DataTyp	:ARRAY[0..79] OF USINT;
		DateTime	:ARRAY[0..79] OF USINT;
		VarName	:ARRAY[0..149] OF USINT;
		y	:UINT;
		status_alloc	:UINT;
		status_free	:UINT;
		temp_status	:UINT;
		PV_xgetadrStatus	:UINT;
		j	:UDINT;
		i	:UDINT;
		FileIdent	:UDINT;
		pFileData	:UDINT;
		Offset	:UDINT;
		OffsetOld	:UDINT;
		CharPerCyclic	:UDINT;
		SpacesCounter	:UDINT;
		Merker	:UDINT;
		SpacesLastRow	:UDINT;
		nextPV	:UDINT;
		Counter	:UDINT;
		PV_Adress	:UDINT;
		data_len	:UDINT;
		FileName	:STRING[80];
		Path	:STRING[80];
		DateTimeStruct	:DTStructure;
		Separator	:USINT;
	END_STRUCT;
			_csv_search_internal : STRUCT
		PV_xgetadrStatus	:UINT;
		PV_ninfoStatus	:UINT;
		PV_itemStatus	:UINT;
		TMP_allocStatus	:UINT;
		Dimension	:UINT;
		ItemNrSoll	:ARRAY[0..49] OF UINT;
		ItemNrIst	:ARRAY[0..49] OF UINT;
		i	:UINT;
		y	:UINT;
		FullStrukturName	:ARRAY[0..299] OF USINT;
		StrukturName	:ARRAY[0..299] OF USINT;
		ArrayName	:ARRAY[0..79] OF USINT;
		UsintArray	:ARRAY[0..79] OF USINT;
		CRLF	:ARRAY[0..2] OF USINT;
		Separator	:ARRAY[0..1] OF USINT;
		Ebene	:USINT;
		Step	:USINT;
		NameCounter	:USINT;
		FoundChar	:USINT;
		Counter_Usint	:USINT;
		Merker	:USINT;
		MerkerArray	:ARRAY[0..49] OF BOOL;
		DataLenght	:UDINT;
		Datatyp	:UDINT;
		PV_Adress	:UDINT;
		Offset	:UDINT;
		TmpValue	:UDINT;
		Lenght	:UDINT;
		Date_and_Time	:DATE_AND_TIME;
		DintTime	:DINT;
		Index	:ARRAY[0..6] OF USINT;
		StartVarName	:ARRAY[0..79] OF USINT;
		VarItemName	:ARRAY[0..299] OF USINT;
		ItemName	:ARRAY[0..79] OF USINT;
		Value	:ARRAY[0..79] OF USINT;
		NextItemReady	:BOOL;
		ArrayStructure	:BOOL;
		ArrayVariable	:BOOL;
		VariableCounter	:UDINT;
	END_STRUCT;
END_TYPE
```
